PROGRAM MAIN
VAR
END_VAR

END_PROGRAM

(* stored: Version 1.1.0.1
   POU MAIN: Id {124ea97a-974a-481e-92b7-de6cac73643a} *)
